(* IEC 61131-3 sources: POMIRTS_lab3/AS/Library_2/ArPnIm, 3 files *)

(* ---- ArPnIm.typ ---- *)
TYPE
	ArPnImSoftwareRevisionType : 	STRUCT
		Prefix : USINT;
		X : USINT;
		Y : USINT;
		Z : USINT;
	END_STRUCT;

	ArPnImIm0Type : 	STRUCT
		VendorID : UINT;
		OrderID : ARRAY[0..19]OF USINT;
		SerialNumber : ARRAY[0..15]OF USINT;
		HardwareRevision : UINT;
		SoftwareRevision : ArPnImSoftwareRevisionType;
		RevisionCounter : UINT;
		ProfileID : UINT;
		ProfileSpecificType : UINT;
		IMVersion : UINT;
		IMSupported : UINT;
	END_STRUCT;

	ArPnImIm5Type : 	STRUCT
		Annotation : ARRAY[0..63]OF USINT;
		OrderID : ARRAY[0..63]OF USINT;
		VendorID : UINT;
		SerialNumber : ARRAY[0..15]OF USINT;
		HardwareRevision : UINT;
		SoftwareRevision : ArPnImSoftwareRevisionType;
	END_STRUCT;

	ArPnImUuidType : STRUCT
		Data : ARRAY[0..15]OF USINT;
	END_STRUCT;

	ArPnImAssetEntryType :
	(
		arPNIM_ASSET_TYPE_FULL := 1,
		arPNIM_ASSET_TYPE_FW_ONLY := 2,
		arPNIM_ASSET_TYPE_HW_ONLY := 3
	);

	ArPnImAssetLevelTreeType : STRUCT
		Levels: ARRAY[0..11]OF UINT;
	END_STRUCT;

	ArPnImAssetSlotSubslotType : STRUCT
		SlotBegin : UINT;
		SubslotBegin : UINT;
		SlotEnd : UINT;
		SubslotEnd : UINT;
	END_STRUCT;

	ArPnImAssetLocationType : STRUCT
		StructureId : USINT;
		LevelTree : ArPnImAssetLevelTreeType;
		SlotSubslot : ArPnImAssetSlotSubslotType;
	END_STRUCT;

	ArPnImAssetDeviceType: STRUCT
		DeviceSubId : UINT;
		DeviceId : UINT;
		VendorId : UINT;
		Organization : UINT;
	END_STRUCT;

	ArPnImAssetDataType: STRUCT
		EntryType : ArPnImAssetEntryType;
		ImUniqueIdentifier : ArPnImUuidType;
		AmLocation : ArPnImAssetLocationType;
		ImAnnotation : ARRAY[0..63]OF USINT;
		ImOrderId : ARRAY[0..63]OF USINT;
		AmSoftwareRev : ARRAY[0..63]OF USINT;
		AmHardwareRev : ARRAY[0..63]OF USINT;
		ImSerialNumber : ARRAY[0..15]OF USINT;
		ImSoftwareRev : ARRAY[0..3]OF USINT;
		AmDeviceIdentification : ArPnImAssetDeviceType;
		AmTypeIdentification : UINT;
		ImHardwareRev : UINT;
	END_STRUCT;

	ArPnImAssetType: STRUCT
		Name : STRING[127];
		ParentName : STRING[127];
		Send : BOOL;
		Valid : BOOL;
		Data : ArPnImAssetDataType;
	END_STRUCT;
END_TYPE

(* ---- ArPnIm.fun ---- *)
{REDUND_CONTEXT} {REDUND_UNREPLICABLE} FUNCTION_BLOCK ArPnImGetDeviceIm0 (*Gets the I&M0 data set for this device*)
	VAR_INPUT
		Execute		: BOOL;					(*Execution of the function block begins on a rising edge of this input.*)
		Device		: STRING[127];			(*Name of the profinet device e.g. SS1.IF1.*)
	END_VAR
	VAR_OUTPUT
		Done		: BOOL;					(*Execution successful. Function block is finished.*)
		Busy 		: BOOL;					(*The function block must continue to be called.*)
		Error		: BOOL;					(*Error occurred during operation.*)
		StatusID	: DINT;  				(*Status information.*)
		Im0 		: ArPnImIm0Type;		(*I&M0 data*)
	END_VAR
	VAR
		Internal	: ARRAY[0..31] OF UDINT; (*Internal variable.*)
	END_VAR
END_FUNCTION_BLOCK

{REDUND_CONTEXT} {REDUND_UNREPLICABLE} FUNCTION_BLOCK ArPnImSetDeviceIdentification (*Sets the device ID and the device type for this device*)
	VAR_INPUT
		Execute		: BOOL;					(*Execution of the function block begins on a rising edge of this input.*)
		Device		: STRING[127];			(*Name of the profinet device e.g. SS1.IF1.*)
		DeviceID	: UINT;					(*Device identification*)
		DeviceType	: ARRAY[0..24]OF USINT;	(*Device type*)
		Im0 		: ArPnImIm0Type;		(*I&M0 data to set*)
	END_VAR
	VAR_OUTPUT
		Done		: BOOL;					(*Execution successful. Function block is finished.*)
		Busy 		: BOOL;					(*The function block must continue to be called.*)
		Error		: BOOL;					(*Error occurred during operation.*)
		StatusID	: DINT;  				(*Status information.*)
	END_VAR
	VAR
		Internal	: ARRAY[0..31] OF UDINT; (*Internal variable.*)
	END_VAR
END_FUNCTION_BLOCK

{REDUND_CONTEXT} {REDUND_UNREPLICABLE} FUNCTION_BLOCK ArPnImSetDeviceIm5 (*Sets the I&M5 data for this device*)
	VAR_INPUT
		Execute		: BOOL;					(*Execution of the function block begins on a rising edge of this input.*)
		Device		: STRING[127];			(*Name of the profinet device e.g. SS1.IF1.*)
		Im5 		: ArPnImIm5Type;		(*I&M5 data to set*)
	END_VAR
	VAR_OUTPUT
		Done		: BOOL;					(*Execution successful. Function block is finished.*)
		Busy 		: BOOL;					(*The function block must continue to be called.*)
		Error		: BOOL;					(*Error occurred during operation.*)
		StatusID	: DINT;  				(*Status information.*)
	END_VAR
	VAR
		Internal	: ARRAY[0..31] OF UDINT; (*Internal variable.*)
	END_VAR
END_FUNCTION_BLOCK

{REDUND_CONTEXT} {REDUND_UNREPLICABLE} FUNCTION_BLOCK ArPnImSetAssets (*Sets asset data for this device*)
	VAR_INPUT
		Execute		: BOOL;					(*Execution of the function block begins on a rising edge of this input.*)
		Device		: STRING[127];			(*Name of the profinet device e.g. SS1.IF1.*)
		AssetArray	: UDINT;				(*Pointer to the asset array.*)
		AssetCount	: UDINT;				(*Number of assets.*)
	END_VAR
	VAR_OUTPUT
		Done		: BOOL;					(*Execution successful. Function block is finished.*)
		Busy 		: BOOL;					(*The function block must continue to be called.*)
		Error		: BOOL;					(*Error occurred during operation.*)
		StatusID	: DINT;  				(*Status information.*)
	END_VAR
	VAR
		Internal	: ARRAY[0..31] OF UDINT; (*Internal variable.*)
	END_VAR
END_FUNCTION_BLOCK

{REDUND_CONTEXT} {REDUND_UNREPLICABLE} FUNCTION_BLOCK ArPnImRemoveAssets (*Removes asset data for this device*)
	VAR_INPUT
		Execute		: BOOL;					(*Execution of the function block begins on a rising edge of this input.*)
		Device		: STRING[127];			(*Name of the profinet device e.g. SS1.IF1.*)
	END_VAR
	VAR_OUTPUT
		Done		: BOOL;					(*Execution successful. Function block is finished.*)
		Busy 		: BOOL;					(*The function block must continue to be called.*)
		Error		: BOOL;					(*Error occurred during operation.*)
		StatusID	: DINT;  				(*Status information.*)
	END_VAR
	VAR
		Internal	: ARRAY[0..31] OF UDINT; (*Internal variable.*)
	END_VAR
END_FUNCTION_BLOCK

{REDUND_CONTEXT} {REDUND_UNREPLICABLE} FUNCTION_BLOCK ArPnImGenerateAssets (*Delivers system-possible assets.*)
	VAR_INPUT
		Execute			: BOOL;					(*Execution of the function block begins on a rising edge of this input.*)
		AssetArray		: UDINT;				(*Pointer to the asset array.*)
		AssetArrayLen	: UDINT;				(*Length of the asset array.*)
	END_VAR
	VAR_OUTPUT
		Done			: BOOL;					(*Execution successful. Function block is finished.*)
		Busy 			: BOOL;					(*The function block must continue to be called.*)
		Error			: BOOL;					(*Error occurred during operation.*)
		StatusID		: DINT;  				(*Status information.*)
		AssetCount		: UDINT;				(*Number of automatically generated assets.*)
	END_VAR
	VAR
		Internal		: ARRAY[0..31] OF UDINT; (*Internal variable.*)
	END_VAR
END_FUNCTION_BLOCK

{REDUND_CONTEXT} {REDUND_UNREPLICABLE} FUNCTION_BLOCK ArPnImGenerateAssetLevels (*Generates the level-tree location information for an array of assets.*)
	VAR_INPUT
		Execute			: BOOL;					(*Execution of the function block begins on a rising edge of this input.*)
		AssetArray		: UDINT;				(*Pointer to the asset array.*)
		AssetCount		: UDINT;				(*Length of the asset array.*)
		StartAsset		: STRING[127];			(*Name of the start asset*)
	END_VAR
	VAR_OUTPUT
		Done			: BOOL;					(*Execution successful. Function block is finished.*)
		Busy 			: BOOL;					(*The function block must continue to be called.*)
		Error			: BOOL;					(*Error occurred during operation.*)
		StatusID		: DINT;  				(*Status information.*)
		InvalidElementIndex : UDINT;			(*Index of the AssetArray element which caused an error.*)
	END_VAR
	VAR
		Internal		: ARRAY[0..31] OF UDINT; (*Internal variable.*)
	END_VAR
END_FUNCTION_BLOCK

{REDUND_CONTEXT} {REDUND_UNREPLICABLE} FUNCTION_BLOCK ArPnImGenerateAssetUuids (*Generates the UUIDs for an array of assets.*)
	VAR_INPUT
		Execute			: BOOL;					(*Execution of the function block begins on a rising edge of this input.*)
		AssetArray		: UDINT;				(*Pointer to the asset array.*)
		AssetCount		: UDINT;				(*Length of the asset array.*)
	END_VAR
	VAR_OUTPUT
		Done			: BOOL;					(*Execution successful. Function block is finished.*)
		Busy 			: BOOL;					(*The function block must continue to be called.*)
		Error			: BOOL;					(*Error occurred during operation.*)
		StatusID		: DINT;  				(*Status information.*)
	END_VAR
	VAR
		Internal		: ARRAY[0..31] OF UDINT; (*Internal variable.*)
	END_VAR
END_FUNCTION_BLOCK

(* ---- ArPnIm.var ---- *)
VAR CONSTANT
	arPNIM_ERR_DEVICE				: DINT := -1070583746;	(*Invalid device name.*)
	arPNIM_ERR_NO_ROOT				: DINT := -1070583745;	(*Invalid root device name*)
	arPNIM_ERR_ASSET_ARRAY			: DINT := -1070583744;	(*Invalid asset array.*)
	arPNIM_ERR_DUPLICATE_ASSET		: DINT := -1070583743;	(*Duplicate asset found.*)
	arPNIM_ERR_FLOATING_ASSET		: DINT := -1070583742;	(*Floating asset found.*)
	arPNIM_ERR_INVALID_START		: DINT := -1070583741;	(*Asset loop found.*)
	arPNIM_ERR_ASSET_DEPTH			: DINT := -1070583740;	(*Asset depth.*)
	arPNIM_ERR_ASSET_NAME			: DINT := -1070583737;	(*Invalid asset name*)

	arPNIM_INF_ARRAY_LEN			: DINT := 1076899952;	(*Array length is to short.*)

	arPNIM_STRUCTURE_ID_LEVEL_TREE		: USINT := 1;
	arPNIM_STRUCTURE_ID_SLOT_SUBSLOT	: USINT := 2;
END_VAR
